// TIA Portal project "Cinta" (V18)

(* hardware
DEVICE "S7-1500/ET200MP station_1"  S7-1500 station
   slot 0: "Rail_0"  Rack  6ES7 590-1***0-0AA0
   slot 1: "PLC_1"  CPU 1516-3 PN/DP  6ES7 516-3AN00-0AB0  V1.8
      slot 3: "CPU display_1"  6ES7591-1BA00-0AA0
      slot 32768: "PROFINET interface_1"  X1
         slot 32769: "Port_1"  X1 P1
         slot 32770: "Port_2"  X1 P2
      slot 33024: "PROFINET interface_2"  X2
         slot 33025: "Port_1"  X2 P1
      slot 33280: "DP interface_1"  X3
   slot 2: "DI 16x24VDC BA_1"  DI 16x24VDC BA  6ES7 521-1BH10-0AA0  V1.1
   slot 3: "DQ 8x24VDC/2A HF_1"  DQ 8x24VDC/2A HF  6ES7 522-1BF00-0AB0  V2.2
   slot 4: "AI 16xI BA_1"  AI 16xI BA  6ES7 531-7MH00-0AB0  V1.0
   slot 5: "AQ 2xU/I ST_1"  AQ 2xU/I ST  6ES7 532-5NB00-0AB0  V1.0
*)

// ===== PLC "PLC_1"  CPU 1516-3 PN/DP =====

FUNCTION_BLOCK "Cinta"   // FB2, STL
TITLE = BLOQUE DE LA CINTA
{ S7_Optimized_Access := 'TRUE' }
VERSION : 0.1
// Este bloque controlará las desconxeiones por petición y error, la conexión, el régimen permanente y las interrupciones de la cinta.
   VAR_INPUT
      PETICION_CONEXION : Bool;   // Petición de conexión de la Cinta.
      PETICION_DESCONEXION : Bool;   // Petición de desconexión de la cinta.
      VELOCIDAD_RAW : Int;   // Entrada de velocidad de la cinta analógica.
      V_med : Real;   // Velocidad deseada en régimen permanente.
      V_MIN : Real;   // Mínimo de velocidad que se puede medir.
      V_MAX : Real;   // Máximo de velocidad que se puede medir.
      V_MAX_ADM : Real;   // Máxima velocidad admitida en régimen permanente.
      V_MIN_ADM : Real;   // Mínima velocidad permitida en régimen permanente.
      SU : Bool;   // Sensor de presencia ultrasonido para detectar las cajas vacías
      PP_A_CINTA : Bool;   // Aviso de que el Pick and Place quiere dejar algo en la cinta.
      DO_NOTHING : Bool;   // Aviso de que la pieza detectada no requiere operación.
      TIEMPO_LIM : Time;   // Tiempo límite de regulación de velocidad.
      TIEMPO_LIM_ERROR_INT : Time;   // Tiempo límite para error de interrupción.
      REARME_LOCAL : Bool;   // Rearme local de la cinta.
      REARME : Bool;   // Rearme global tras emergencia asíncrona.
      EMER : Bool;   // Emergencia asíncrona.
      MANT : Bool;   // Petición de congelación de la cinta por mantenimiento.
      APAGADO_CONFIRMADO : Bool;   // Apagado de la cinta confirmado.
      ERROR_AUTO_DIAG : Bool;   // Error encontrado en el autodiagnóstico.
      CINTA_OK : Bool;   // Autodiagnóstico correcto.
   END_VAR
   VAR_OUTPUT
      M_ACELERAR : Bool;   // Señal de aceleración del motor.
      M_FRENAR : Bool;   // Señal de frenada del motor.
      M_PARAR : Bool;   // Señal de parada suave mediante rampa de frenado.
      PARADA_ASINCRONA : Bool;   // Señal de parada brusca por emergecia asíncrona.
      PARADA_SINCRONA : Bool;   // Señal de parada brusca por emergencia síncrona..
      CINTA_ON : Bool;   // Acuse de recibo de puesta en marcha.
      CINTA_OFF : Bool;   // Acuse de recibo de apagado.
      CINTA_CONG : Bool;   // Acuse de recibo de parada por mantenimiento.
      AUTO_DIAG_CINTA : Bool;   // Señal de autodiagnóstico de la cinta
      CINTA_APAGAR : Bool;   // Orden de apagado de la cinta.
      ERROR_GLOBAL : Bool;   // Chivato de error global.
      ERROR_LOCAL : Bool;   // Chivato de error local.
   END_VAR
   VAR
      B_TRABAJO : Bool;   // Bit que indica si la cinta ya estaba encendida.
      X_ERROR_LOCAL : Bool;   // Etapa pozo por error local.
      X_EMER_GLOBAL : Bool;   // Etapa pozo por emergencia global.
      X1 : Bool;   // Etapa de autodiagnóstico.
      X2 : Bool;   // Etapa de aceleración inicial.
      X3 : Bool;   // Régimen permanente de velocidad.
      X4 : Bool;   // Etapa de frenado.
      X5 : Bool;   // Etapa de aceleración.
      XM1 : Bool;   // Macroetapa de interrupción por nueva pieza.
      XM2 : Bool;   // Macroetapa de interrupción por pieza terminadad.
      X10 : Bool;   // Etapa de solicitud a la desconexión natural.
      X_FIN : Bool;   // Apagado de la cinta.
      ERROR_PARADA : Bool;   // Error durante la parada de la cinta.
      C_FIN_INT1 : Bool;   // Conector para el fin de la interrupción 1.
      C_INI_INT2 : Bool;   // Conector para el inicio de la interrupción 2.
      ERROR_TEMPORIZACION : Bool;   // Error debido a exceso de tiempo.
      ERROR_MEDICION : Bool;   // Error durante la medición de la velocidad.
      Marcha_Motor_X2 : "Marcha_Motor";
      Marcha_Motor_X4 : "Marcha_Motor";
      Marcha_Motor_X5 : "Marcha_Motor";
      Marcha_Motor_PARADA : "Marcha_Motor";
      Interrupcion_PIEZA_NUEVA : "Interrupcion";
      Interrupcion_PIEZA_TERMINADA : "Interrupcion";
   END_VAR
   VAR_TEMP
      V_baja : Bool;   // La velocidad es muy lenta.
      V_alta : Bool;   // La velocidad es muy rápida.
      V_parada : Bool;   // Está parado.
      V_REAL : Real;   // Valor convertido de la velocidad.
      V_OK_SUBIDA : Bool;   // Velocidad alcanzada acelerando.
      V_OK_BAJADA : Bool;   // Velocidad alcanzada frenando.
      FIN_INT : Bool;   // Fin interrupción.
      FIN_MAN : Bool;   // Fin de la maniobra.
      FIN_PARADA : Bool;   // Fin de la parada.
   END_VAR
BEGIN

REGION Network 1: DESCONEXIÓN NORMAL
   // Desconexión de la cinta porque no se ha encendido todavía.
         AN    #PETICION_CONEXION;

         R     #B_TRABAJO;

         R     #CINTA_OFF;
         R     #CINTA_ON;
         R     #AUTO_DIAG_CINTA;

         JCN   _DESCONEXION;

         CALL  #Marcha_Motor_X2
         ( RESET        := TRUE,
           FIN_MANIOBRA := ,
           TIEMPO_LIM   := ,
           MOTOR        := #M_ACELERAR,
           B_FIN        := ,
           ERROR_TIEMPO :=
         );

         CALL  #Marcha_Motor_X4
         ( RESET        := TRUE,
           FIN_MANIOBRA := ,
           TIEMPO_LIM   := ,
           MOTOR        := #M_FRENAR,
           B_FIN        := ,
           ERROR_TIEMPO :=
         );

         CALL  #Marcha_Motor_X5
         ( RESET        := TRUE,
           FIN_MANIOBRA := ,
           TIEMPO_LIM   := ,
           MOTOR        := #M_ACELERAR,
           B_FIN        := ,
           ERROR_TIEMPO :=
         );

         CALL  #Marcha_Motor_PARADA
         ( RESET        := TRUE,
           FIN_MANIOBRA := ,
           TIEMPO_LIM   := ,
           MOTOR        := #CINTA_APAGAR,
           B_FIN        := ,
           ERROR_TIEMPO :=
         );

         CALL  #Interrupcion_PIEZA_NUEVA
         ( RESET            := TRUE,
           C_PARADA         := ,
           FIN_INTERRUPCION := ,
           TIEMPO_LIM       := ,
           M_PARAR          := #M_PARAR,
           B_FIN            := ,
           ERROR_PARADA     := ,
           M_ACELERAR       := #M_ACELERAR
         );

         CALL  #Interrupcion_PIEZA_TERMINADA
         ( RESET            := TRUE,
           C_PARADA         := ,
           FIN_INTERRUPCION := ,
           TIEMPO_LIM       := ,
           M_PARAR          := #M_PARAR,
           B_FIN            := ,
           ERROR_PARADA     := ,
           M_ACELERAR       := #M_ACELERAR
         );


   _DESCONEXION:NOP   0;
END_REGION

REGION Network 2: DESCONEXIÓN POR EMERGENCIA GLOBAL
         A     #X_EMER_GLOBAL;

         S     #PARADA_ASINCRONA;
         S     #ERROR_GLOBAL;
         R     #PARADA_SINCRONA;
         R     #CINTA_OFF;
         R     #CINTA_ON;
         R     #AUTO_DIAG_CINTA;

         JCN   _ERRGL;

         CALL  #Marcha_Motor_X2
         ( RESET        := TRUE,
           FIN_MANIOBRA := ,
           TIEMPO_LIM   := ,
           MOTOR        := #M_ACELERAR,
           B_FIN        := ,
           ERROR_TIEMPO :=
         );

         CALL  #Marcha_Motor_X4
         ( RESET        := TRUE,
           FIN_MANIOBRA := ,
           TIEMPO_LIM   := ,
           MOTOR        := #M_FRENAR,
           B_FIN        := ,
           ERROR_TIEMPO :=
         );

         CALL  #Marcha_Motor_X5
         ( RESET        := TRUE,
           FIN_MANIOBRA := ,
           TIEMPO_LIM   := ,
           MOTOR        := #M_ACELERAR,
           B_FIN        := ,
           ERROR_TIEMPO :=
         );

         CALL  #Marcha_Motor_PARADA
         ( RESET        := TRUE,
           FIN_MANIOBRA := ,
           TIEMPO_LIM   := ,
           MOTOR        := #CINTA_APAGAR,
           B_FIN        := ,
           ERROR_TIEMPO :=
         );

         CALL  #Interrupcion_PIEZA_NUEVA
         ( RESET            := TRUE,
           C_PARADA         := ,
           FIN_INTERRUPCION := ,
           TIEMPO_LIM       := ,
           M_PARAR          := #M_PARAR,
           B_FIN            := ,
           ERROR_PARADA     := ,
           M_ACELERAR       := #M_ACELERAR
         );

         CALL  #Interrupcion_PIEZA_TERMINADA
         ( RESET            := TRUE,
           C_PARADA         := ,
           FIN_INTERRUPCION := ,
           TIEMPO_LIM       := ,
           M_PARAR          := #M_PARAR,
           B_FIN            := ,
           ERROR_PARADA     := ,
           M_ACELERAR       := #M_ACELERAR
         );



   _ERRGL:NOP   0;
END_REGION

REGION Network 3: DESCONEXION ERROR LOCAL
   // Desconexión debida a un error local en la cinta, ya sea por el control de velocidad o durante el autodiagnóstico.
         A     #X_ERROR_LOCAL;

         R     #PARADA_ASINCRONA;
         S     #ERROR_LOCAL;
         S     #PARADA_SINCRONA;
         R     #CINTA_OFF;
         R     #CINTA_ON;
         R     #AUTO_DIAG_CINTA;

         JCN   _ERRLO;

         CALL  #Marcha_Motor_X2
         ( RESET        := TRUE,
           FIN_MANIOBRA := ,
           TIEMPO_LIM   := ,
           MOTOR        := #M_ACELERAR,
           B_FIN        := ,
           ERROR_TIEMPO :=
         );

         CALL  #Marcha_Motor_X4
         ( RESET        := TRUE,
           FIN_MANIOBRA := ,
           TIEMPO_LIM   := ,
           MOTOR        := #M_FRENAR,
           B_FIN        := ,
           ERROR_TIEMPO :=
         );

         CALL  #Marcha_Motor_X5
         ( RESET        := TRUE,
           FIN_MANIOBRA := ,
           TIEMPO_LIM   := ,
           MOTOR        := #M_ACELERAR,
           B_FIN        := ,
           ERROR_TIEMPO :=
         );

         CALL  #Marcha_Motor_PARADA
         ( RESET        := TRUE,
           FIN_MANIOBRA := ,
           TIEMPO_LIM   := ,
           MOTOR        := #CINTA_APAGAR,
           B_FIN        := ,
           ERROR_TIEMPO :=
         );

         CALL  #Interrupcion_PIEZA_NUEVA
         ( RESET            := TRUE,
           C_PARADA         := ,
           FIN_INTERRUPCION := ,
           TIEMPO_LIM       := ,
           M_PARAR          := #M_PARAR,
           B_FIN            := ,
           ERROR_PARADA     := ,
           M_ACELERAR       := #M_ACELERAR
         );

         CALL  #Interrupcion_PIEZA_TERMINADA
         ( RESET            := TRUE,
           C_PARADA         := ,
           FIN_INTERRUPCION := ,
           TIEMPO_LIM       := ,
           M_PARAR          := #M_PARAR,
           B_FIN            := ,
           ERROR_PARADA     := ,
           M_ACELERAR       := #M_ACELERAR
         );



   _ERRLO:NOP   0;
END_REGION

REGION Network 4: CONEXIÓN
         A     #PETICION_CONEXION;
         FP    #B_TRABAJO;

         S     #X1;
         R     #X2;
         R     #X3;
         R     #X4;
         R     #X5;
         R     #XM1;
         R     #XM2;
         R     #X10;
         R     #X_EMER_GLOBAL;
         R     #X_ERROR_LOCAL;
         R     #X_FIN;

         R     #ERROR_MEDICION;
         R     #ERROR_PARADA;
         R     #ERROR_TEMPORIZACION;

         R     #PARADA_ASINCRONA;
         R     #PARADA_SINCRONA;
         R     #ERROR_GLOBAL;
         R     #ERROR_LOCAL;
         R     #AUTO_DIAG_CINTA;
         R     #CINTA_OFF;
         R     #CINTA_ON;

         JCN   _CONEXION;

         CALL  #Marcha_Motor_X2
         ( RESET        := TRUE,
           FIN_MANIOBRA := ,
           TIEMPO_LIM   := ,
           MOTOR        := #M_ACELERAR,
           B_FIN        := ,
           ERROR_TIEMPO :=
         );

         CALL  #Marcha_Motor_X4
         ( RESET        := TRUE,
           FIN_MANIOBRA := ,
           TIEMPO_LIM   := ,
           MOTOR        := #M_FRENAR,
           B_FIN        := ,
           ERROR_TIEMPO :=
         );

         CALL  #Marcha_Motor_X5
         ( RESET        := TRUE,
           FIN_MANIOBRA := ,
           TIEMPO_LIM   := ,
           MOTOR        := #M_ACELERAR,
           B_FIN        := ,
           ERROR_TIEMPO :=
         );

         CALL  #Marcha_Motor_PARADA
         ( RESET        := TRUE,
           FIN_MANIOBRA := ,
           TIEMPO_LIM   := ,
           MOTOR        := #CINTA_APAGAR,
           B_FIN        := ,
           ERROR_TIEMPO :=
         );

         CALL  #Interrupcion_PIEZA_NUEVA
         ( RESET            := TRUE,
           C_PARADA         := ,
           FIN_INTERRUPCION := ,
           TIEMPO_LIM       := ,
           M_PARAR          := #M_PARAR,
           B_FIN            := ,
           ERROR_PARADA     := ,
           M_ACELERAR       := #M_ACELERAR
         );

         CALL  #Interrupcion_PIEZA_TERMINADA
         ( RESET            := TRUE,
           C_PARADA         := ,
           FIN_INTERRUPCION := ,
           TIEMPO_LIM       := ,
           M_PARAR          := #M_PARAR,
           B_FIN            := ,
           ERROR_PARADA     := ,
           M_ACELERAR       := #M_ACELERAR
         );



   _CONEXION:NOP   0;
END_REGION

REGION Network 5: CONGELACIÓN
   // Congelación de la cinta por matenimiento.
         A     #MANT;

         =     #CINTA_CONG;
         R     #AUTO_DIAG_CINTA;

         JCN   _CONGELACION;

         CALL  #Marcha_Motor_X2
         ( RESET        := TRUE,
           FIN_MANIOBRA := ,
           TIEMPO_LIM   := ,
           MOTOR        := #M_ACELERAR,
           B_FIN        := ,
           ERROR_TIEMPO :=
         );

         CALL  #Marcha_Motor_X4
         ( RESET        := TRUE,
           FIN_MANIOBRA := ,
           TIEMPO_LIM   := ,
           MOTOR        := #M_FRENAR,
           B_FIN        := ,
           ERROR_TIEMPO :=
         );

         CALL  #Marcha_Motor_X5
         ( RESET        := TRUE,
           FIN_MANIOBRA := ,
           TIEMPO_LIM   := ,
           MOTOR        := #M_ACELERAR,
           B_FIN        := ,
           ERROR_TIEMPO :=
         );

         CALL  #Marcha_Motor_PARADA
         ( RESET        := TRUE,
           FIN_MANIOBRA := ,
           TIEMPO_LIM   := ,
           MOTOR        := #CINTA_APAGAR,
           B_FIN        := ,
           ERROR_TIEMPO :=
         );

         CALL  #Interrupcion_PIEZA_NUEVA
         ( RESET            := TRUE,
           C_PARADA         := ,
           FIN_INTERRUPCION := ,
           TIEMPO_LIM       := ,
           M_PARAR          := #M_PARAR,
           B_FIN            := ,
           ERROR_PARADA     := ,
           M_ACELERAR       := #M_ACELERAR
         );

         CALL  #Interrupcion_PIEZA_TERMINADA
         ( RESET            := TRUE,
           C_PARADA         := ,
           FIN_INTERRUPCION := ,
           TIEMPO_LIM       := ,
           M_PARAR          := #M_PARAR,
           B_FIN            := ,
           ERROR_PARADA     := ,
           M_ACELERAR       := #M_ACELERAR
         );


   _CONGELACION:NOP   0;

         A     #MANT;
         BEC;
END_REGION

REGION Network 6: REARME GLOBAL
   // Rearme tras emergencia global.
         A     #X_EMER_GLOBAL;
         A     #REARME;

         R     #X_EMER_GLOBAL;
         R     #B_TRABAJO;
END_REGION

REGION Network 7: REARME LOCAL
   // Rearme tras emergencia local.
   // Se coloca antes que el segmento de desconexión por emergencia global para que se salte y entre directamente al segmento de conexión.
         A     #X_ERROR_LOCAL;
         A     #REARME_LOCAL;

         R     #X_ERROR_LOCAL;
         R     #B_TRABAJO;
END_REGION

REGION Network 8: CONECTORES
   // Tratamiento de todos los conectores necesarios (velocidad y tiempos límite).
         CALL  "Tratamiento_velocidad"
         ( V_RAW       := #VELOCIDAD_RAW,
           V_med       := #V_med,
           V_MIN       := #V_MIN,
           V_MAX       := #V_MAX,
           V_MAX_ADM   := #V_MAX_ADM,
           V_MIN_ADM   := #V_MIN_ADM,
           V_baja      := #V_baja,
           V_alta      := #V_alta,
           V_parada    := #V_parada,
           V_OK_SUBIDA := #V_OK_SUBIDA,
           V_OK_BAJADA := #V_OK_BAJADA,
           V_REAL      := #V_REAL,
           ERROR       := #ERROR_MEDICION
         );

   // Conector de fin de interrupción 1
         AN    #SU;
         O     #DO_NOTHING;
         =     #C_FIN_INT1;

   // Conector de inicio de interrupción 2
         AN    #SU;
         A     #PP_A_CINTA;
         =     #C_INI_INT2;
END_REGION

REGION Network 9: ERROR GLOBAL
   // Salto a etapa de emergencia global.
         A     #EMER;

         S     #X_EMER_GLOBAL;
         R     #X1;
         R     #X2;
         R     #X3;
         R     #X4;
         R     #X5;
         R     #XM1;
         R     #XM2;
END_REGION

REGION Network 10: ERROR LOCAL
   // Salto a etapa de emergencia local.
         A     #ERROR_AUTO_DIAG;
         O     #ERROR_MEDICION;
         O     #ERROR_PARADA;
         O     #ERROR_TEMPORIZACION;
         O(;
         A     #X3;
         A     #V_parada;
         );

         S     #X_ERROR_LOCAL;
         R     #XM1;
         R     #XM2;
         R     #X1;
         R     #X2;
         R     #X3;
         R     #X4;
         R     #X5;
END_REGION

REGION Network 11: CINTA ENCENDIDA (X1 -> X2)
   // La cinta se pone en marcha tras el autodiagnóstico.
         A     #X1;
         A     #CINTA_OK;

         S     #X2;
         R     #X1;
END_REGION

REGION Network 12: X2 -> X3
   // La cinta llega al régimen permanente
         A     #X2;

         JCN   _X2;

         CALL  #Marcha_Motor_X2
         ( RESET        := FALSE,
           FIN_MANIOBRA := #V_OK_SUBIDA,
           TIEMPO_LIM   := #TIEMPO_LIM,
           MOTOR        := #M_ACELERAR,
           B_FIN        := #FIN_MAN,
           ERROR_TIEMPO := #ERROR_TEMPORIZACION
         );

         A     #FIN_MAN;
         S     #X3;
         R     #X2;

   _X2:  NOP   0;
END_REGION

REGION Network 13: X3 -> X4
   // La cinta pierde velocidad.
         A     #X3;
         A     #V_alta;

         S     #X4;
         R     #X3;
END_REGION

REGION Network 14: X3 -> X5
   // La cinta gana velocidad.
         A     #X3;
         A     #V_baja;

         S     #X5;
         R     #X3;
END_REGION

REGION Network 15: X4 -> X3
   // Vuelta al régimen permanente.
         A     #X4;
         JCN   _X4;

         CALL  #Marcha_Motor_X4
         ( RESET        := FALSE,
           FIN_MANIOBRA := #V_OK_BAJADA,
           TIEMPO_LIM   := #TIEMPO_LIM,
           MOTOR        := #M_FRENAR,
           B_FIN        := #FIN_MAN,
           ERROR_TIEMPO := #ERROR_TEMPORIZACION
         );

         A     #FIN_MAN;
         S     #X3;
         R     #X4;

   _X4:  NOP   0;
END_REGION

REGION Network 16: X5 ->X3
   // Vuelta al régimen permanente.
         A     #X5;
         JCN   _X5;

         CALL  #Marcha_Motor_X5
         ( RESET        := FALSE,
           FIN_MANIOBRA := #V_OK_SUBIDA,
           TIEMPO_LIM   := #TIEMPO_LIM,
           MOTOR        := #M_ACELERAR,
           B_FIN        := #FIN_MAN,
           ERROR_TIEMPO := #ERROR_TEMPORIZACION
         );

         A     #FIN_MAN;
         S     #X3;
         R     #X5;

   _X5:  NOP   0;
END_REGION

REGION Network 17: INTERRUPCION 1 (XM1)
         A(;
         O     #X2;
         O     #X3;
         O     #X4;
         O     #X5;
         );
         A     #SU;

         S     #XM1;
         R     #X2;
         R     #X3;
         R     #X4;
         R     #X5;
END_REGION

REGION Network 18: TRATAMIENTO DE INTERRUPCION 1 (XM1)
         A     #XM1;

         JCN   _INTERRUPCION_1;

   // Interrumpir los procesos que se estén ejecutando
         CALL  #Marcha_Motor_X2
         ( RESET        := TRUE,
           FIN_MANIOBRA := ,
           TIEMPO_LIM   := ,
           MOTOR        := #M_ACELERAR,
           B_FIN        := ,
           ERROR_TIEMPO :=
         );

         CALL  #Marcha_Motor_X4
         ( RESET        := TRUE,
           FIN_MANIOBRA := ,
           TIEMPO_LIM   := ,
           MOTOR        := #M_FRENAR,
           B_FIN        := ,
           ERROR_TIEMPO :=
         );

         CALL  #Marcha_Motor_X5
         ( RESET        := TRUE,
           FIN_MANIOBRA := ,
           TIEMPO_LIM   := ,
           MOTOR        := #M_ACELERAR,
           B_FIN        := ,
           ERROR_TIEMPO :=
         );

   // Ejecutar la interrupción
         CALL  #Interrupcion_PIEZA_NUEVA
         ( RESET            := FALSE,
           C_PARADA         := #V_parada,
           FIN_INTERRUPCION := #C_FIN_INT1,
           TIEMPO_LIM       := #TIEMPO_LIM_ERROR_INT,
           M_PARAR          := #M_PARAR,
           B_FIN            := #FIN_INT,
           ERROR_PARADA     := #ERROR_PARADA,
           M_ACELERAR       := #M_ACELERAR
         );

         A     #FIN_INT;

         S     #X2;
         R     #XM1;

         A     #ERROR_PARADA;

         S     #X_ERROR_LOCAL;
         R     #XM1;

   _INTERRUPCION_1:NOP   0;
END_REGION

REGION Network 19: INTERRUPCION 2 (XM2)
         A(;
         O     #X2;
         O     #X3;
         O     #X4;
         O     #X5;
         );
         A     #C_INI_INT2;

         S     #XM2;
         R     #X2;
         R     #X3;
         R     #X4;
         R     #X5;
END_REGION

REGION Network 20: TRATAMIENTO DE INTERRUPCION 2 (XM2)
         A     #XM2;

         JCN   _INTERRUPCION_2;

   // Interrumpir los procesos que se estén ejecutando
         CALL  #Marcha_Motor_X2
         ( RESET        := TRUE,
           FIN_MANIOBRA := ,
           TIEMPO_LIM   := ,
           MOTOR        := #M_ACELERAR,
           B_FIN        := ,
           ERROR_TIEMPO :=
         );

         CALL  #Marcha_Motor_X4
         ( RESET        := TRUE,
           FIN_MANIOBRA := ,
           TIEMPO_LIM   := ,
           MOTOR        := #M_FRENAR,
           B_FIN        := ,
           ERROR_TIEMPO :=
         );

         CALL  #Marcha_Motor_X5
         ( RESET        := TRUE,
           FIN_MANIOBRA := ,
           TIEMPO_LIM   := ,
           MOTOR        := #M_ACELERAR,
           B_FIN        := ,
           ERROR_TIEMPO :=
         );

   // Ejecutar la interrupción
         CALL  #Interrupcion_PIEZA_TERMINADA
         ( RESET            := FALSE,
           C_PARADA         := #V_parada,
           FIN_INTERRUPCION := #SU,
           TIEMPO_LIM       := #TIEMPO_LIM_ERROR_INT,
           M_PARAR          := #M_PARAR,
           B_FIN            := #FIN_INT,
           ERROR_PARADA     := #ERROR_PARADA,
           M_ACELERAR       := #M_ACELERAR
         );

         A     #FIN_INT;

         S     #X2;
         R     #XM2;

         A     #ERROR_PARADA;

         S     #X_ERROR_LOCAL;
         R     #XM2;

   _INTERRUPCION_2:NOP   0;
END_REGION

REGION Network 21: PETICION DE PARADA
         A     #PETICION_DESCONEXION;
         A(;
         O     #X1;
         O     #X2;
         O     #X3;
         O     #X4;
         O     #X5;
         );

         S     #X10;
         R     #X1;
         R     #X2;
         R     #X3;
         R     #X4;
         R     #X5;
END_REGION

REGION Network 22: TRATAMIENTO X1
         A     #X1;
         =     #AUTO_DIAG_CINTA;
         S     #CINTA_ON;
END_REGION

REGION Network 23: APAGADO DE LA CINTA.
         A     #X10;
         S     #CINTA_OFF;
         R     #CINTA_ON;
         JCN   _PARADA;

         CALL  #Marcha_Motor_X2
         ( RESET        := TRUE,
           FIN_MANIOBRA := ,
           TIEMPO_LIM   := ,
           MOTOR        := #M_ACELERAR,
           B_FIN        := ,
           ERROR_TIEMPO :=
         );

         CALL  #Marcha_Motor_X4
         ( RESET        := TRUE,
           FIN_MANIOBRA := ,
           TIEMPO_LIM   := ,
           MOTOR        := #M_FRENAR,
           B_FIN        := ,
           ERROR_TIEMPO :=
         );

         CALL  #Marcha_Motor_X5
         ( RESET        := TRUE,
           FIN_MANIOBRA := ,
           TIEMPO_LIM   := ,
           MOTOR        := #M_ACELERAR,
           B_FIN        := ,
           ERROR_TIEMPO :=
         );

         CALL  #Marcha_Motor_PARADA
         ( RESET        := FALSE,
           FIN_MANIOBRA := #APAGADO_CONFIRMADO,
           TIEMPO_LIM   := #TIEMPO_LIM,
           MOTOR        := #CINTA_APAGAR,
           B_FIN        := #FIN_PARADA,
           ERROR_TIEMPO := #ERROR_TEMPORIZACION
         );

         A     #FIN_PARADA;
         S     #X_FIN;
         R     #X10;

         A     #ERROR_TEMPORIZACION;
         S     #X_ERROR_LOCAL;
         R     #X10;

   _PARADA:NOP   0;
END_REGION
END_FUNCTION_BLOCK

// folder: Cinta

FUNCTION_BLOCK "Interrupcion"   // FB1, STL
TITLE = Bloque de interrupción en la cinta
{ S7_Optimized_Access := 'TRUE' }
VERSION : 0.1
// Esta secuencia se ejecutará siempre que el robot Pick and Place quiera coger o dejar una pieza en la cinta.
   VAR_INPUT
      RESET : Bool;   // Evento asíncrono de prioridad máxima para la desconexión del bloque.
      C_PARADA : Bool;   // Indica que la cinta está completamente parada. Se recomienda que sea un sensor de velocidad que marque 0.
      FIN_INTERRUPCION : Bool;   // Indica que la interrupción ha finalizado y se vuelve al ciclo normal.
      TIEMPO_LIM : Time;   // Tiempo límite para la parada, si se sobrepasa dará error.
   END_VAR
   VAR_OUTPUT
      M_PARAR : Bool;   // Para la cinta de forma suave, con una rampa de frenado.
      B_FIN : Bool;   // Indica el fin de la interrupción y vuelta al ciclo normal.
      ERROR_PARADA : Bool;   // Indica que la cinta ha tardado mucho en parar. Ha habido un error.
      M_ACELERAR : Bool;   // Acelerar el motor.
   END_VAR
   VAR
      B_TRABAJO : Bool;   // Bit de trabajo que controla la consexión por flanco
      X_PARADA : Bool;   // Etapa en la que se realiza la rampa de frenado.
      X_ESPERA : Bool;   // Etapa de espera hasta el fin de la interrupción.
      X_MOTOR : Bool;   // Etapa en la que se acelera el motor para evitar que se vuelva a tratar la misma pieza.
      AVISO_ERROR : Bool;   // Aviso interno del error de parada por tiempo excesivo.
      TEMP_ALTO : Bool;   // Salto del temporizador.
      MOTOR_OK : Bool;   // El motor ha movido la pieza lo suficiente.
      X_FIN : Bool;   // Etapa de fin de la interrupción.
      IEC_Timer_Parada : TON_TIME;
      IEC_Timer_0_MOTOR : TON_TIME;
      T : Time;
   END_VAR
BEGIN

REGION Network 1: DESCONEXIÓN POR RESET
   // Evento asíncrono de prioridad máxima. Resetea el bloque y sale de él.
         A     #RESET;

         R     #B_TRABAJO;
         R     #AVISO_ERROR;
         R     #X_ESPERA;
         R     #X_PARADA;
         R     #X_MOTOR;
         R     #X_FIN;

         R     #M_PARAR;
         R     #M_ACELERAR;
         R     #B_FIN;
         R     #ERROR_PARADA;

         JCN   _RESET;
         CALL  RESET_TIMER
         ( "TIMER" := #IEC_Timer_Parada
         );

         CALL  RESET_TIMER
         ( "TIMER" := #IEC_Timer_0_MOTOR
         );

   _RESET:NOP   0;

         A     #RESET;
         BEC;
END_REGION

REGION Network 2: DESCONEXIÓN POR ERROR DE TIEMPO
   // Evento síncrono de error por temporización
         A     #AVISO_ERROR;

         R     #B_TRABAJO;

         S     #ERROR_PARADA;

         R     #M_PARAR;
         R     #M_ACELERAR;

         JCN   _TIEMPO;
         CALL  RESET_TIMER
         ( "TIMER" := #IEC_Timer_Parada
         );

         CALL  RESET_TIMER
         ( "TIMER" := #IEC_Timer_0_MOTOR
         );

   _TIEMPO:NOP   0;

         A     #AVISO_ERROR;
         R     #AVISO_ERROR;
         BEC;
END_REGION

REGION Network 3: DESCONEXIÓN POR FIN DE LA INTERRUPCIÓN
   // Fin de la interrupción natural.
         A     #X_FIN;

         R     #B_TRABAJO;

         S     #B_FIN;

         R     #M_PARAR;
         R     #M_ACELERAR;

         JCN   _FIN;
         CALL  RESET_TIMER
         ( "TIMER" := #IEC_Timer_Parada
         );

         CALL  RESET_TIMER
         ( "TIMER" := #IEC_Timer_0_MOTOR
         );

   _FIN: NOP   0;

         A     #X_FIN;
         R     #X_FIN;
         BEC;
END_REGION

REGION Network 4: CONEXIÓN DE LA INTERRUPCIÓN
         SET;
         FP    #B_TRABAJO;

         S     #X_PARADA;
         R     #X_FIN;
         R     #X_ESPERA;
         R     #X_MOTOR;
         R     #AVISO_ERROR;

         R     #ERROR_PARADA;
         R     #B_FIN;
END_REGION

REGION Network 5: ACTIVACIÓN DEL ERROR POR TIEMPO
   // Si se está demasiado tiempo en la etapa de parada se activa el aviso de error y se ejecuta la desconexión. 
   // No es necesario limpiar este temporizador explícitamente ya que lo hace automáticamente cuando el evento de disparo está a FALSE.
         CALL  #IEC_Timer_Parada
         ( IN := #X_PARADA,
           PT := #TIEMPO_LIM,
           Q  := #TEMP_ALTO,
           ET := #T
         );


         A     #TEMP_ALTO;
         S     #AVISO_ERROR;
END_REGION

REGION Network 6: CONTROL DEL TIEMPO DEL MOTOR
   // Se mide el tiempo necesario para que la pieza deje de estar delante del sensor y pueda volver al régimen permanente.
   // Se trata de un tiempo fijo no modificable, por lo que se pone directamente.
         CALL  #IEC_Timer_0_MOTOR
         ( IN := #X_MOTOR,
           PT := T#5s,
           Q  := #MOTOR_OK,
           ET :=
         );
END_REGION

REGION Network 7: PASO A ESPERA
   // Paso a la etapa de espera si la cinta se ha parado.
         A     #X_PARADA;
         A     #C_PARADA;

         S     #X_ESPERA;
         R     #X_PARADA;
END_REGION

REGION Network 8: PASO A MOVIMIENTO
   // Una vez a terminado la acción se mueve la cinta para evitar tratar de nuevo la misma pieza
         A     #X_ESPERA;
         A     #FIN_INTERRUPCION;

         S     #X_MOTOR;
         R     #X_ESPERA;
END_REGION

REGION Network 9: PASO A FIN
   // Paso a la etapa de fin si la interrupción se ha terminado.
         A     #X_MOTOR;
         A     #MOTOR_OK;

         S     #X_FIN;
         R     #X_MOTOR;
END_REGION

REGION Network 10: TRATAMIENTO DE LA PARADA
   // Tratamiento de la etapa de parada.
         A     #X_PARADA;
         =     #M_PARAR;
END_REGION

REGION Network 11: TRATAMIENTO DEL MOVIMIENTO
   // Tratamiento de la etapa de movimiento.
         A     #X_MOTOR;
         =     #M_ACELERAR;
END_REGION
END_FUNCTION_BLOCK

FUNCTION_BLOCK "Marcha_Motor"   // FB3, STL
TITLE = Bloque de velocidad en la cinta
{ S7_Optimized_Access := 'TRUE' }
VERSION : 0.1
// Esta secuencia se ejecutará siempre que la cinta deba moderar la velocidad.
   VAR_INPUT
      RESET : Bool;   // Evento asíncrono de prioridad máxima para la desconexión del bloque.
      FIN_MANIOBRA : Bool;   // Indica que la maniobra ha finalizado y se vuelve al ciclo normal.
      TIEMPO_LIM : Time;   // Tiempo límite para la maniobra, si se sobrepasa dará error.
   END_VAR
   VAR_OUTPUT
      MOTOR : Bool;   // Actúa sobre el motor.
      B_FIN : Bool;   // Indica el fin de la maniobra y vuelta al ciclo normal.
      ERROR_TIEMPO : Bool;   // Indica que la cinta ha tardado mucho en parar. Ha habido un cambiar su velocidad.
   END_VAR
   VAR
      B_TRABAJO : Bool;   // Bit de trabajo que controla la consexión por flanco
      X_MARCHA : Bool;   // Etapa en la que se realiza la acción.
      AVISO_ERROR : Bool;   // Aviso interno del error de parada por tiempo excesivo.
      TEMP_ALTO : Bool;   // Salto del temporizador.
      X_FIN : Bool;   // Etapa de fin de la interrupción.
      IEC_Timer_Marcha : TON_TIME;
   END_VAR
BEGIN

REGION Network 1: DESCONEXIÓN POR RESET
   // Evento asíncrono de prioridad máxima. Resetea el bloque y sale de él.
         A     #RESET;

         R     #B_TRABAJO;
         R     #AVISO_ERROR;
         R     #X_MARCHA;
         R     #X_FIN;

         R     #MOTOR;
         R     #B_FIN;
         R     #ERROR_TIEMPO;

         JCN   _RESET;
         CALL  RESET_TIMER
         ( "TIMER" := #IEC_Timer_Marcha
         );
   _RESET:NOP   0;

         A     #RESET;
         BEC;
END_REGION

REGION Network 2: DESCONEXIÓN POR ERROR DE TIEMPO
   // Evento síncrono de error por temporización
         A     #AVISO_ERROR;

         R     #B_TRABAJO;

         S     #ERROR_TIEMPO;

         R     #MOTOR;

         JCN   _TIEMPO;
         CALL  RESET_TIMER
         ( "TIMER" := #IEC_Timer_Marcha
         );
   _TIEMPO:NOP   0;

         A     #AVISO_ERROR;
         R     #AVISO_ERROR;
         BEC;
END_REGION

REGION Network 3: DESCONEXIÓN POR FIN DE LA MARCHA
   // Fin de la marcha natural.
         A     #X_FIN;

         R     #B_TRABAJO;

         S     #B_FIN;

         R     #MOTOR;

         JCN   _FIN;
         CALL  RESET_TIMER
         ( "TIMER" := #IEC_Timer_Marcha
         );
   _FIN: NOP   0;

         A     #X_FIN;
         R     #X_FIN;
         BEC;
END_REGION

REGION Network 4: CONEXIÓN DE LA MARCHA
         SET;
         FP    #B_TRABAJO;

         S     #X_MARCHA;
         R     #X_FIN;
         R     #AVISO_ERROR;

         R     #ERROR_TIEMPO;
         R     #B_FIN;
END_REGION

REGION Network 5: ACTIVACIÓN DEL ERROR POR TIEMPO
   // Si se está demasiado tiempo en la etapa de parada se activa el aviso de error y se ejecuta la desconexión.
         CALL  #IEC_Timer_Marcha
         ( IN := #X_MARCHA,
           PT := #TIEMPO_LIM,
           Q  := #TEMP_ALTO,
           ET :=
         );


         A     #TEMP_ALTO;
         S     #AVISO_ERROR;
END_REGION

REGION Network 6: PASO A FIN
   // Paso a la etapa de fin si la interrupción se ha terminado.
         A     #X_MARCHA;
         A     #FIN_MANIOBRA;

         S     #X_FIN;
         R     #X_MARCHA;
END_REGION

REGION Network 7: TRATAMIENTO DE LA MARCHA
   // Tratamiento de la etapa de parada.
         A     #X_MARCHA;
         =     #MOTOR;
END_REGION
END_FUNCTION_BLOCK

FUNCTION "Tratamiento_velocidad" : Void   // FC1, STL
TITLE = Conectores de la señal analógica.
{ S7_Optimized_Access := 'TRUE' }
VERSION : 0.1
// En este bloque se comparará la velocidad del motor con la que debería tener.
   VAR_INPUT
      V_RAW : Int;   // Valor de la señal desde el sensor.
      V_med : Real;   // Velocidad permanente que se quiere comparar.
      V_MIN : Real;   // Mínimo de velocidad que se puede medir.
      V_MAX : Real;   // Máximo de velocidad que se puede medir.
      V_MAX_ADM : Real;   // Máxima velocidad admitida en régimen permanente.
      V_MIN_ADM : Real;   // Mínima velocidad permitida en régimen permanente.
   END_VAR
   VAR_OUTPUT
      V_baja : Bool;   // La velocidad es muy lenta.
      V_alta : Bool;   // La velocidad es muy rápida.
      V_parada : Bool;   // Está parado.
      V_OK_SUBIDA : Bool;   // Velocidad alcanzada acelerando.
      V_OK_BAJADA : Bool;   // Velocidad alcanzada frenando.
   END_VAR
   VAR_IN_OUT
      V_REAL : Real;   // Velocidad real del motor.
      ERROR : Bool;   // Error durante la medición.
   END_VAR
BEGIN

REGION Network 1: Tratamiento de la señal analógica.
   // Conversión dela señal medida por el sensor.
         CALL  "Tratamiento_analogico"
         ( raw_vel     := #V_RAW,
           V_min       := #V_MIN,
           V_max       := #V_MAX,
           V           := #V_REAL,
           aviso_error := #ERROR
         );
END_REGION

REGION Network 2: Error durante la medición.
   // Si hay un error en la medición se sale del bloque.
         A     #ERROR;
         BEC;
END_REGION

REGION Network 3: Comparación de velocidades.
   // Se compara si la velocidad es baja.
         L     #V_REAL;
         L     #V_MIN_ADM;
         <R;
         =     #V_baja;
END_REGION

REGION Network 4: Comparación de velocidades.
   // Se compara si la velocidad es alta.
         L     #V_REAL;
         L     #V_MAX_ADM;
         >R;
         =     #V_alta;
END_REGION

REGION Network 5: Comparación de velocidades.
   // Se compara si la velocidad es 0.
         L     #V_REAL;
         L     0.0;
         ==R;
         =     #V_parada;
END_REGION

REGION Network 6: Velocidad OK de subida.
   // Se ha acelerado al régimen aceptable.
         L     #V_REAL;
         L     #V_med;
         >R;
         =     #V_OK_SUBIDA;
END_REGION

REGION Network 7: Velocidad OK de bajada.
   // Se ha frenado al régimen aceptable.
         A     <0;
         =     #V_OK_BAJADA;
END_REGION
END_FUNCTION

// folder: Globales

FUNCTION "Tratamiento_analogico" : Void   // FC2, STL
TITLE = TRATAMIENTO ANALÓGICO
{ S7_Optimized_Access := 'TRUE' }
VERSION : 0.1
// Este bloque se encarga del tratamiento de la señal analógica.
   VAR_INPUT
      raw_vel : Int;   // Velocidad digitalizada del sensor.
      V_min : Real;   // Mínimo de velocidad que se puede medir.
      V_max : Real;   // Máximo de velocidad que se puede medir.
   END_VAR
   VAR_OUTPUT
      V : Real;   // Velocidad analógica convertida.
      aviso_error : Bool;   // Error durante tratamiento.
   END_VAR
   VAR_TEMP
      ret_val_1 : Word;   // Error.
   END_VAR
BEGIN

REGION Network 1: SEÑAL ANALÓGICA
   // Conversión de la señal de entrada a un valor real.
         CALL  SCALE
         ( IN      := #raw_vel,
           HI_LIM  := #V_max,
           LO_LIM  := #V_min,
           BIPOLAR := FALSE,
           RET_VAL := #ret_val_1,
           OUT     := #V
         );
END_REGION

REGION Network 2: GESTIÓN DEL ERROR
   // Si ret_val_1 es 0, la medida es correcta. Si no da error.
         L     #ret_val_1;
         L     0;
         <>I;
         =     #aviso_error;
END_REGION
END_FUNCTION